FUNCTION FindOldest : myPersonType
VAR_INPUT
	ListOfEmplyees:myEmployees;
END_VAR
VAR
	i: INT;
END_VAR

FindOldest:=ListOfEmplyees[1];
FOR	i:=2	TO	SIZEOF(ListOfEmplyees)/SIZEOF(myPersonType)	DO
	IF	ListOfEmplyees[i].age>0	THEN
		IF	ListOfEmplyees[i].age>FindOldest.age	THEN
			FindOldest:=ListOfEmplyees[i];
		END_IF
	END_IF
END_FOR

END_FUNCTION

(* stored: Version 1.1.0.1, ProductVersion 3.1.4024.11
   POU FindOldest: Id {7da3d37c-72f7-4f0f-a2ec-d27607693613}, SpecialFunc None *)
